// TIA Portal V20 export
TYPE "LBP_typeMcp310CPnOutput"
TITLE = MCP 310C PN image / Image du MCP 310C PN
// Output image of MCP 310C PN / Image de sortie du MCP 310C PN
   STRUCT
      standard { S7_SetPoint := 'True'} : "LBP_typeMcp310StandardOutput";   // Output image of MCP 310 / Image de sortie du MCP 310
   END_STRUCT;
END_TYPE
